FUNCTION_BLOCK Grade_Equipamentos (* Composite Function Block Type *)
  (* Standard: 61499-2 *)
  (* Version 0.0, 2/24/2026, template *)
  PACKAGE Hidryco.HidrycoLib;
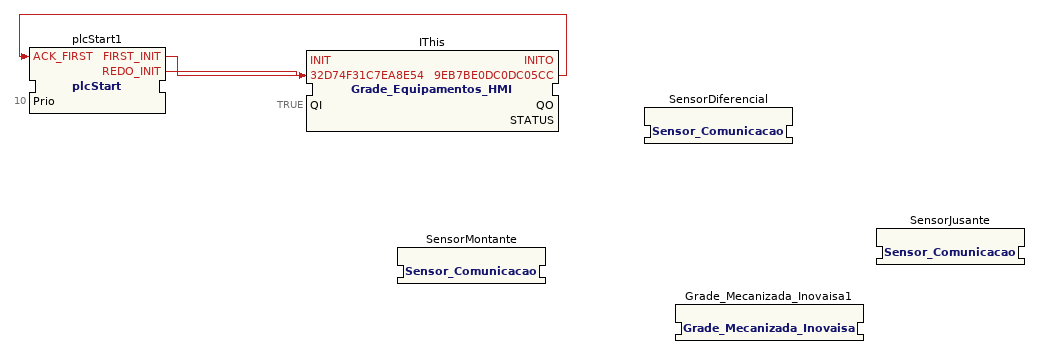
  FBS
    SensorMontante : Sensor_Comunicacao;
    SensorDiferencial : Sensor_Comunicacao;
    SensorJusante : Sensor_Comunicacao;
    IThis : Grade_Equipamentos_HMI(QI := TRUE);
    plcStart1 : plcStart(Prio := 10);
    Grade_Mecanizada_Inovaisa1 : Grade_Mecanizada_Inovaisa;
  END_FBS
  EVENT_CONNECTIONS
    plcStart1.FIRST_INIT TO IThis.32D74F31C7EA8E54;
    plcStart1.REDO_INIT TO IThis.32D74F31C7EA8E54;
    IThis.9EB7BE0DC0DC05CC TO plcStart1.ACK_FIRST;
  END_CONNECTIONS
END_FUNCTION_BLOCK
